FUNCTION_BLOCK HVAC_B28_CM_CALL
VAR_INPUT
END_VAR
VAR_OUTPUT
END_VAR
VAR
	AI_1_Temp : PlantAndCMs.CM_SensorAnalog_V2;
	AI_2_Pres: PlantAndCMs.CM_SensorAnalog_V2;
	
	AI_DMP_1: PlantAndCMs.CM_SensorAnalog_V2;
	
	AV_1 : PlantAndCMs.CM_Actuator2State_V2;
	AV_2 : PlantAndCMs.CM_Actuator2State_V2;
	
	MTR_1 : PlantAndCMs.CM_AO_V2;
	MTR_2 : PlantAndCMs.CM_AO_V2;
	
	DMP_1 : PlantAndCMs.CM_AO_V2;
	
	
	
	DMP_2 : PlantAndCMs.CM_AO_V2;
	
END_VAR

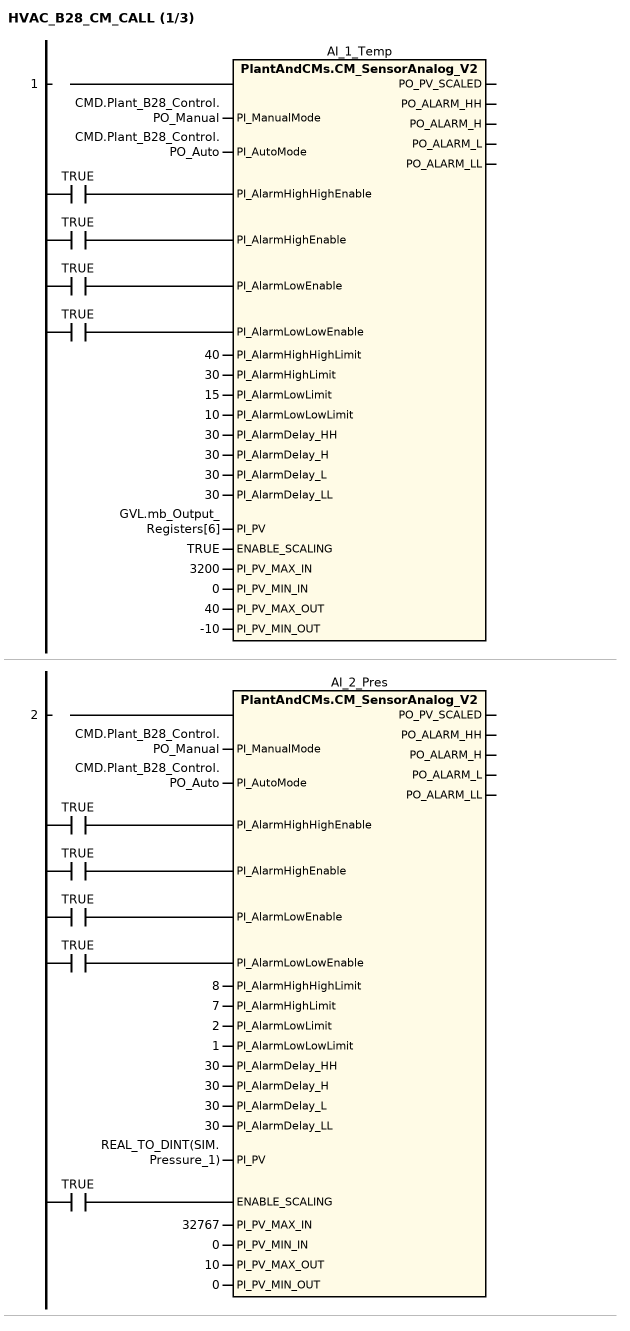
// NETWORK 1
AI_1_Temp(
    PI_ManualMode := CMD.Plant_B28_Control.PO_Manual,
    PI_AutoMode := CMD.Plant_B28_Control.PO_Auto,
    PI_AlarmHighHighEnable := TRUE,
    PI_AlarmHighEnable := TRUE,
    PI_AlarmLowEnable := TRUE,
    PI_AlarmLowLowEnable := TRUE,
    PI_AlarmHighHighLimit := 40,
    PI_AlarmHighLimit := 30,
    PI_AlarmLowLimit := 15,
    PI_AlarmLowLowLimit := 10,
    PI_AlarmDelay_HH := 30,
    PI_AlarmDelay_H := 30,
    PI_AlarmDelay_L := 30,
    PI_AlarmDelay_LL := 30,
    PI_PV := GVL.mb_Output_Registers[6],
    ENABLE_SCALING := TRUE,
    PI_PV_MAX_IN := 3200,
    PI_PV_MIN_IN := 0,
    PI_PV_MAX_OUT := 40,
    PI_PV_MIN_OUT := -10); // PlantAndCMs.CM_SensorAnalog_V2

// NETWORK 2
AI_2_Pres(
    PI_ManualMode := CMD.Plant_B28_Control.PO_Manual,
    PI_AutoMode := CMD.Plant_B28_Control.PO_Auto,
    PI_AlarmHighHighEnable := TRUE,
    PI_AlarmHighEnable := TRUE,
    PI_AlarmLowEnable := TRUE,
    PI_AlarmLowLowEnable := TRUE,
    PI_AlarmHighHighLimit := 8,
    PI_AlarmHighLimit := 7,
    PI_AlarmLowLimit := 2,
    PI_AlarmLowLowLimit := 1,
    PI_AlarmDelay_HH := 30,
    PI_AlarmDelay_H := 30,
    PI_AlarmDelay_L := 30,
    PI_AlarmDelay_LL := 30,
    PI_PV := REAL_TO_DINT(SIM.Pressure_1),
    ENABLE_SCALING := TRUE,
    PI_PV_MAX_IN := 32767,
    PI_PV_MIN_IN := 0,
    PI_PV_MAX_OUT := 10,
    PI_PV_MIN_OUT := 0); // PlantAndCMs.CM_SensorAnalog_V2

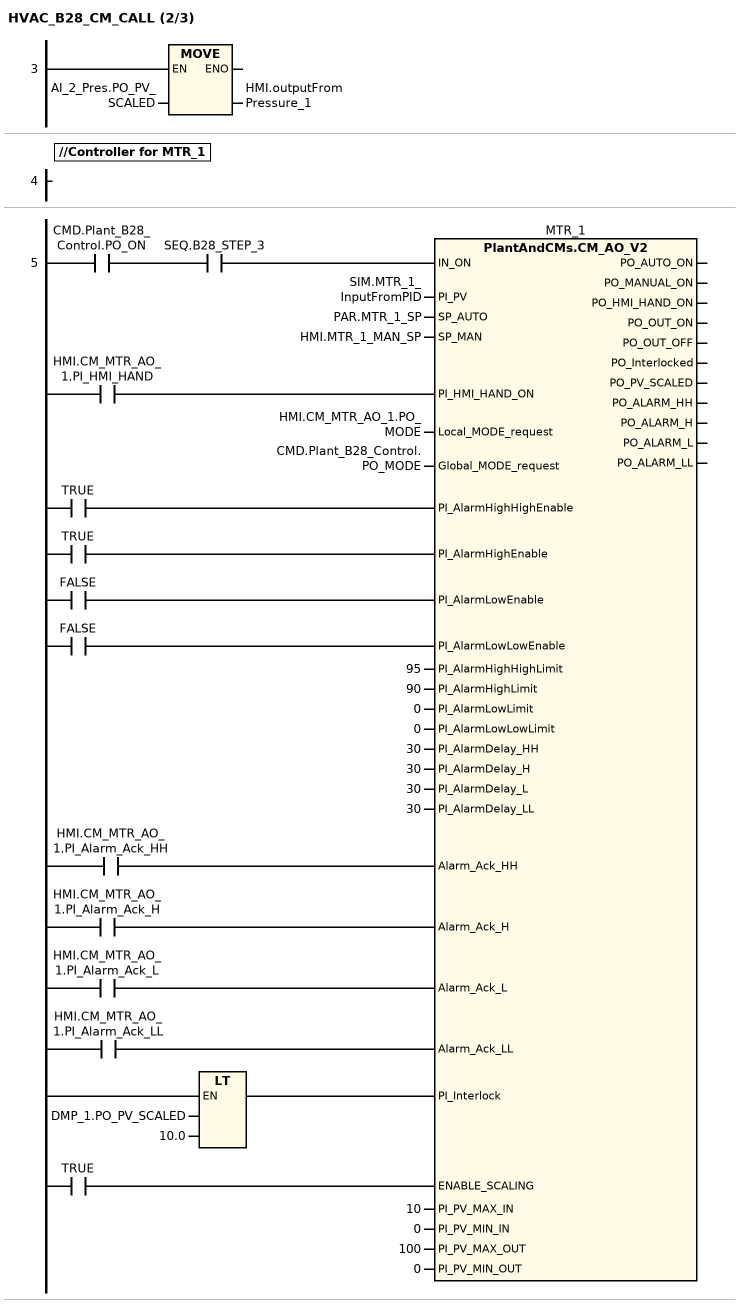
// NETWORK 3
HMI.outputFromPressure_1 := AI_2_Pres.PO_PV_SCALED;

// NETWORK 4
// label: //Controller for MTR_1

// NETWORK 5
MTR_1(
    IN_ON := CMD.Plant_B28_Control.PO_ON AND SEQ.B28_STEP_3,
    PI_PV := SIM.MTR_1_InputFromPID,
    SP_AUTO := PAR.MTR_1_SP,
    SP_MAN := HMI.MTR_1_MAN_SP,
    PI_HMI_HAND_ON := HMI.CM_MTR_AO_1.PI_HMI_HAND,
    Local_MODE_request := HMI.CM_MTR_AO_1.PO_MODE,
    Global_MODE_request := CMD.Plant_B28_Control.PO_MODE,
    PI_AlarmHighHighEnable := TRUE,
    PI_AlarmHighEnable := TRUE,
    PI_AlarmLowEnable := FALSE,
    PI_AlarmLowLowEnable := FALSE,
    PI_AlarmHighHighLimit := 95,
    PI_AlarmHighLimit := 90,
    PI_AlarmLowLimit := 0,
    PI_AlarmLowLowLimit := 0,
    PI_AlarmDelay_HH := 30,
    PI_AlarmDelay_H := 30,
    PI_AlarmDelay_L := 30,
    PI_AlarmDelay_LL := 30,
    Alarm_Ack_HH := HMI.CM_MTR_AO_1.PI_Alarm_Ack_HH,
    Alarm_Ack_H := HMI.CM_MTR_AO_1.PI_Alarm_Ack_H,
    Alarm_Ack_L := HMI.CM_MTR_AO_1.PI_Alarm_Ack_L,
    Alarm_Ack_LL := HMI.CM_MTR_AO_1.PI_Alarm_Ack_LL,
    PI_Interlock := DMP_1.PO_PV_SCALED < 10.0,
    ENABLE_SCALING := TRUE,
    PI_PV_MAX_IN := 10,
    PI_PV_MIN_IN := 0,
    PI_PV_MAX_OUT := 100,
    PI_PV_MIN_OUT := 0); // PlantAndCMs.CM_AO_V2

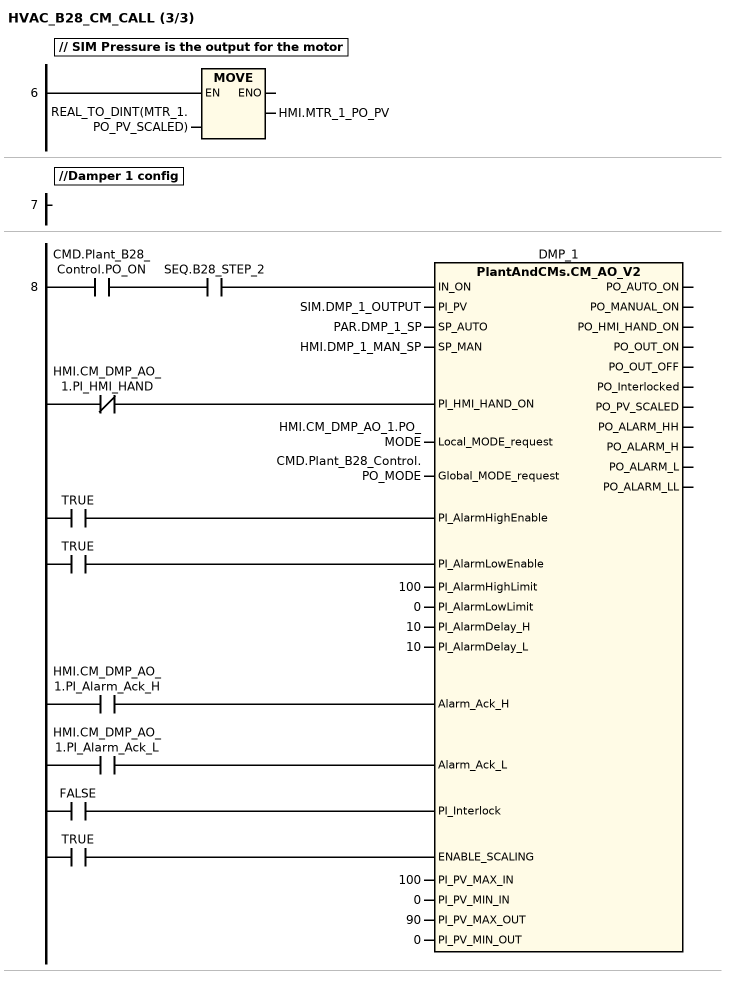
// NETWORK 6
// label: // SIM Pressure is the output for the motor
HMI.MTR_1_PO_PV := REAL_TO_DINT(MTR_1.PO_PV_SCALED);

// NETWORK 7
// label: //Damper 1 config

// NETWORK 8
DMP_1(
    IN_ON := CMD.Plant_B28_Control.PO_ON AND SEQ.B28_STEP_2,
    PI_PV := SIM.DMP_1_OUTPUT,
    SP_AUTO := PAR.DMP_1_SP,
    SP_MAN := HMI.DMP_1_MAN_SP,
    PI_HMI_HAND_ON := NOT HMI.CM_DMP_AO_1.PI_HMI_HAND,
    Local_MODE_request := HMI.CM_DMP_AO_1.PO_MODE,
    Global_MODE_request := CMD.Plant_B28_Control.PO_MODE,
    PI_AlarmHighEnable := TRUE,
    PI_AlarmLowEnable := TRUE,
    PI_AlarmHighLimit := 100,
    PI_AlarmLowLimit := 0,
    PI_AlarmDelay_H := 10,
    PI_AlarmDelay_L := 10,
    Alarm_Ack_H := HMI.CM_DMP_AO_1.PI_Alarm_Ack_H,
    Alarm_Ack_L := HMI.CM_DMP_AO_1.PI_Alarm_Ack_L,
    PI_Interlock := FALSE,
    ENABLE_SCALING := TRUE,
    PI_PV_MAX_IN := 100,
    PI_PV_MIN_IN := 0,
    PI_PV_MAX_OUT := 90,
    PI_PV_MIN_OUT := 0); // PlantAndCMs.CM_AO_V2

END_FUNCTION_BLOCK

(* stored: Version 1.1.0.1, ProductVersion 3.1.4024.13
   POU HVAC_B28_CM_CALL: Id {63a8426a-4f5f-4f88-91ff-83b944a9acdc}, SpecialFunc None *)
